(* IEC 61131-3 sources: SHU_NSTV/src/lib/Interfaces, 3 files *)

(* ---- BasicControl.st ---- *)
INTERFACE BasicControl

METHOD Set_Power
VAR_INPUT
	x : BOOL;
END_VAR

PROPERTY Power : BOOL
(*
* 	Чтобы получить выходной сигнал из функционального блока, требуется вызвать свойство Power.
*	Значение Power можно присовить, например, на питание контактора исполнительного механизма.	-	-	-	-	-	-	-	-	: PU1_KM_cmdOn := PU1.Power;
*	Чтобы получить сигнал работы от механизма, требуется записать сигнал механизма в свойство Power	-	-	-	-	-	-	-	: PU1.Power := PU1_KM_On;
*																																^
*	Важно: Логика функционального блока подразумевает, что свойство Power будет присвоено на питание контактора,				^
*	а сигнал работы исполнительного механизма (статус: включён) будет присовен внутрь свойства Power. Как показано на примере выше.
*)

(* ---- BasicControl_OpenClose.st ---- *)
INTERFACE BasicControl_OpenClose
METHOD Close
VAR_INPUT
END_VAR

METHOD Open
VAR_INPUT
END_VAR

METHOD Stop
VAR_INPUT
END_VAR

(* ---- BasicControlCommands.st ---- *)
INTERFACE BasicControlCommands

METHOD Start
VAR_INPUT
	access : BOOL;
	device : BasicControl;
END_VAR

METHOD Stop
VAR_INPUT
	access: BOOL;
	device : BasicControl;
END_VAR
